(* PLC project Generated.project, CODESYS CODESYS V3.5 SP19 Patch 1 *)
(* stored: creationDateTime 2026-09-06T13:00:42.383652, modificationDateTime 2026-09-06T13:00:42.383652 *)

(* ======================================================================= 🧩 ST_Fault — Brique socle défaut (2 vues : live + latchée) ─────────────────────────────────────────────────────────────── 🎯 Rôle : porter l'état défaut d'un composant, applicable dans TOUS les cas (acquittable ou non), sans brique warning séparée. • Vue LIVE (Error / ErrorId) : suit la cause, retombe seule à 0. • Vue LATCHÉE (Latched / LatchedId): mémorisée au défaut, reste jusqu'au front Reset. Le choix acquittable / non-acquittable se fait PAR CAUSE (ST_FaultCause.Latching), jamais par bloc. 🔒 Sécurité : interlock TOUJOURS sur la cause brute (Error / ErrorId), jamais sur l'acquittement. Reset TOUJOURS effectif, jamais conditionné (std §9). 🧬 Composition : brique de base réutilisable — sortie de FB, struct métier, GVL. Texte IHM NON stocké ici : dérivé côté IHM depuis LatchedId / ErrorId. 📄 Doc : DOC/STDS/CODE_QUALITY_STANDARDS.md §2quinquies / §9 ======================================================================= *)
TYPE ST_Fault : STRUCT
  Error : BOOL;  (* <-- [DIAG] vue LIVE : au moins une cause présente maintenant *)
  ErrorId : WORD;  (* <-- [DIAG] bitfield des causes présentes maintenant (0 si aucune) *)
  Latched : BOOL;  (* <-- [DIAG] vue LATCHÉE : défaut non acquitté, reste jusqu'au front Reset *)
  LatchedId : WORD;  (* <-- [DIAG] ErrorId figé à l'apparition du défaut, effacé au Reset *)
END_STRUCT;
END_TYPE

(* ======================================================================= 🧩 ST_FaultCause — Cause élémentaire alimentant ST_Fault (socle FB_FaultCore) ─────────────────────────────────────────────────────────────── 🎯 Rôle : une cause exprimée EN CLAIR (BOOL + libellé), sans bitfield ni masque. Le FB métier remplit une liste (ARRAY[0..15] OF ST_FaultCause) ; le socle FB_FaultCore en déduit ST_Fault (vue live + vue latchée). 🔒 Sécurité : interlock TOUJOURS sur Active (cause brute), jamais sur le latch. Latching = TRUE → la cause ARME la vue latchée (défaut à acquitter). Latching = FALSE → la cause n'alimente que la vue live (retombe seule). Fail-safe : une cause laissée à Latching=FALSE reste visible en live — pour la rendre acquittable, il faut le déclarer explicitement. 📄 Doc : DOC/STDS/CODE_QUALITY_STANDARDS.md §2quinquies / §9 ======================================================================= *)
TYPE ST_FaultCause : STRUCT
  Active : BOOL;  (* 1 = cause présente maintenant (interlock sur cette valeur) *)
  Latching : BOOL;  (* 1 = cause à acquitter (arme Latched) ; 0 = live seulement *)
  Texte : STRING;  (* libellé prêt IHM (non stocké dans ST_Fault, dérivé côté IHM) *)
END_STRUCT;
END_TYPE

(* ======================================================================= 🔌 FB_Encoder_Abs — Acquisition codeur absolu (accès bus EtherCAT) ─────────────────────────────────────────────────────────────── 🎯 Rôle : Accès bus EtherCAT, extraction positions brutes et séquence de Preset SDO 🔒 Polarité : EncoderAvailable=TRUE si communication bus et esclave OK 🔌 Architecture : Module d'acquisition codeur absolu 📄 Doc métier : DOC/AF/AF_Partie-09_Fonction_Encoder_v2.4.md ======================================================================= === DECLARATION (à coller dans la partie déclaration du POU FB_Encoder_Abs) === *)
FUNCTION_BLOCK FB_Encoder_Abs
  VAR_INPUT
    Enable : BOOL;  (* === COMMANDES & AUTORISATIONS === --> [CMD] Autorisation generale FB (TRUE=Autorise) *)
    Reset : BOOL;  (* --> [CMD] Acquittement defaut (front montant) *)
    PresetRequest : BOOL;  (* --> [CMD] Demande de preset (front montant) *)
    RawPosIn : UDINT;  (* === BUS ETHERCAT & CAPTEUR HW === --> [HW] Position brute EtherCAT *)
    AlarmsIn : UINT;  (* --> [HW] Codes alarmes bruts EtherCAT *)
    WarningsIn : UINT;  (* --> [HW] Codes avertissements bruts EtherCAT *)
    SlaveOperational : BOOL;  (* --> [HW] Statut esclave EtherCAT operationnel *)
    PointsPerRev : UDINT := 8192;  (* === PARAMETRES & REGLAGES === --> [CFG] Resolution codeur (pts/tour) *)
    PresetValue : UDINT;  (* --> [CFG] Valeur cible de preset *)
    PresetTimeout : TIME := TIME#2s0ms;  (* --> [CFG] Temporisation max attente preset *)
    PresetTolerancePts : UDINT := 10;  (* --> [CFG] Tolerance relecture post-preset (pts) *)
  END_VAR
  VAR_OUTPUT
    Ready : BOOL;  (* === ETATS IEC & SYNOPTIQUE === <-- [STAT] FB pret a fonctionner *)
    Fault : ST_Fault;  (* 🧩 Statut transverse (forme cible ST_Fault) *)
    RawPos : UDINT;  (* === MESURES & DONNEES CODEUR === <-- [DIAG] Position brute gelee si non disponible *)
    EncoderAvailable : BOOL;  (* <-- [STAT] Codeur operationnel et disponible *)
    AngleRaw : UINT;  (* <-- [DIAG] Angle brut sur un tour (MOD PointsPerRev) *)
    TurnCount : UDINT;  (* <-- [DIAG] Nombre de tours bruts (RawPos / PointsPerRev) *)
    PresetTriggerCmd : WORD;  (* === COMMANDES & ECHANGE BUS ETHERCAT === <-- [ACT] Ordre declenchement preset vers PDO Rx *)
    CodeSeqTriggerCmd : WORD;  (* <-- [ACT] Ordre sequence code vers PDO Rx *)
    PresetValueOut : UDINT;  (* <-- [ACT] Valeur de preset transmise au PDO Rx *)
  END_VAR
  VAR
    ResetEdge : R_TRIG;  (* === DETECTEURS DE FRONT === . [LOC] Detecteur front montant Reset *)
    PresetReqEdge : R_TRIG;  (* . [LOC] Detecteur front montant PresetRequest *)
    PresetTimer : TON;  (* === TEMPORISATEURS INTERNES === . [LOC] Temporisateur timeout sequence preset *)
    PresetTimerVisual : TON;  (* . [LOC] Temporisateur maintien visuel impulsion (500ms) *)
    PresetSeqStep : INT;  (* === VARIABLES INTERNES DE CALCUL & ETAT === . [LOC] Etape sequence preset (0:IDLE, 1:PULSE/WAIT) *)
    RawDiff : DINT;  (* . [LOC] Ecart signe entre RawPos et PresetValueOut *)
    PresetCompleted : BOOL;  (* . [LOC] Fait de fin de maintien preset (un scan) *)
    PresetTimeoutError : BOOL;  (* . [LOC] Latch interne timeout séquence preset *)
    instFault : FB_FaultCore;  (* === SOCLE DEFAUT (FB_FaultCore) === * [INST] Socle défaut transverse *)
    instCauses : ARRAY[0..15] OF ST_FaultCause;  (* . [LOC] Table des causes nommées *)
  END_VAR

            

// === IMPLEMENTATION (à coller dans le corps ST du POU FB_Encoder_Abs) ===

{region "§1 Causes & Socle Défaut (évalué en continu)"}
// 🔑 1. RESET FRONT
ResetEdge(CLK := Reset);

// 🔍 2. DIAGNOSTIC BUS / ALARME (Cause 0 : live)
instCauses[0].Active   := (AlarmsIn <> 0) OR NOT SlaveOperational;
instCauses[0].Latching := FALSE;
instCauses[0].Texte    := 'Defaut communication EtherCAT codeur absolu';

// ⏱️ 3. TIMEOUT PRESET (Cause 1 : latched)
IF ResetEdge.Q AND (PresetSeqStep = 0) THEN
    PresetTimeoutError := FALSE;
END_IF;
instCauses[1].Active   := PresetTimeoutError;
instCauses[1].Latching := TRUE;
instCauses[1].Texte    := 'Timeout sequence preset SDO codeur';

// Appel du socle de défaut
instFault(Enable := Enable, Reset := Reset, Causes := instCauses);
Fault := instFault.Fault;

EncoderAvailable := NOT instCauses[0].Active;
{endregion}

{region "§2 Gate neutralisation"}
// 🛑 2. GATE
IF NOT Enable THEN
    EncoderAvailable := FALSE;
    Ready := FALSE;
    PresetTriggerCmd := 0; CodeSeqTriggerCmd := 0; PresetValueOut := 0;
    PresetSeqStep := 0;
    PresetCompleted := FALSE;
    PresetTimer(IN := FALSE, PT := PresetTimeout);
    PresetTimerVisual(IN := FALSE, PT := T#500MS);
    // RawPos, AngleRaw et TurnCount sont volontairement gelés hors Enable
    // (AF09 F09.01 / AC5) : aucune lecture bus ni remise a zero dans ce gate.
    RETURN;
END_IF;

Ready := Enable AND NOT Fault.Latched;
{endregion}

{region "§3 Lecture position"}
// 📥 3. LECTURE POSITION — GELER SUR DOUTE (Partie10 §6)
// Si EncoderAvailable=FALSE : RawPos/AngleRaw/TurnCount conservent leur dernière valeur (pas de RETURN
// global ici pour ne pas geler aussi la séquence preset/l'état — seule la lecture est gelée).
IF EncoderAvailable THEN
    RawPos := RawPosIn;   // Sens de comptage géré côté codeur (CoE 6000h bit0, startup parameter CODESYS) — voir Partie10 §3bis. Plus de calcul ici.
    AngleRaw := UDINT_TO_UINT(RawPos MOD PointsPerRev);
    TurnCount := RawPos / PointsPerRev;
END_IF;
{endregion}

{region "§4 Séquence preset"}
// 🔧 4. SÉQUENCE PRESET (écriture bus)
// PresetTriggerCmd := 2 déclenche le référencement à PresetValue (valeur de commande, pas un
// masque de bits). CodeSeqTriggerCmd : rôle non identifié — laissé à 0, PAS piloté tant que sa
// fonction n'est pas confirmée. Ne jamais lui donner une valeur arbitraire.
PresetReqEdge(CLK := PresetRequest);
PresetCompleted := FALSE;
CodeSeqTriggerCmd := 0;                 // non piloté — rôle inconnu, voir note ci-dessus
CASE PresetSeqStep OF
    0: // IDLE
        PresetTriggerCmd := 0;
        IF PresetReqEdge.Q AND EncoderAvailable THEN
            PresetValueOut := PresetValue;
            PresetSeqStep := 1;
            PresetTimer(IN := TRUE, PT := PresetTimeout);
        END_IF;
    1: // Déclenchement preset (laissé actif pendant 0.5s pour confort visuel en simulation/bus)
        PresetTriggerCmd := 2;   // Référence le codeur à PresetValueOut
        RawDiff := UDINT_TO_DINT(RawPos) - UDINT_TO_DINT(PresetValueOut);
        IF ABS(RawDiff) <= UDINT_TO_DINT(PresetTolerancePts) THEN
            PresetTimer(IN := FALSE, PT := PresetTimeout);
            PresetTimerVisual(IN := TRUE, PT := T#500MS);
            IF PresetTimerVisual.Q THEN
                PresetTriggerCmd := 0;
                PresetCompleted := TRUE;
                PresetSeqStep := 0;
                PresetTimerVisual(IN := FALSE, PT := T#500MS);
            END_IF;
        ELSIF PresetTimer.Q THEN
            PresetTriggerCmd := 0;
            PresetTimeoutError := TRUE;
            PresetSeqStep := 0;
            PresetTimer(IN := FALSE, PT := PresetTimeout);
            PresetTimerVisual(IN := FALSE, PT := T#500MS);
        END_IF;
END_CASE;
{endregion}

          
END_FUNCTION_BLOCK

(* ======================================================================= 🧩 FB_FaultCore — Socle de remplissage de ST_Fault (vue live + vue latchée) ─────────────────────────────────────────────────────────────── 🎯 Rôle : à partir d'une LISTE de causes en clair (ARRAY[0..15] OF ST_FaultCause), produire la brique ST_Fault : • Error / ErrorId : vue LIVE, suit les causes Active, retombe seule. • Latched / LatchedId: vue LATCHÉE, chaque bit figé à l'apparition d'une cause `Active AND Latching`, conservé jusqu'au front Reset. 🔒 Sécurité : - interlock TOUJOURS sur `Causes[i].Active` (cause brute), jamais sur le latch. - Reset TOUJOURS effectif, jamais conditionné (std §9) — agit même Enable=FALSE. - Latching=FALSE → cause visible en LIVE seulement (fail-safe : reste visible). - un défaut laté non acquitté reste publié même FB désactivé (pas d'effacement silencieux sur bascule Enable OFF→ON sans Reset). - une cause à acquitter réapparue re-arme son bit (ré-alarme). 🧬 Un seul socle, réutilisé par tout FB `standard` qui expose un ST_Fault. Pas de State, pas de Warning, pas de texte — hors périmètre de ce socle. 📄 Doc : DOC/STDS/CODE_QUALITY_STANDARDS.md §2quinquies / §9 ======================================================================= *)
FUNCTION_BLOCK FB_FaultCore
  VAR_INPUT
    Enable : BOOL;  (* --> [CMD] Autorisation générale du FB porteur *)
    Reset : BOOL;  (* --> [CMD] Front d'acquittement (jamais conditionné, §9) *)
    Causes : ARRAY[0..15] OF ST_FaultCause;  (* --> [CMD] Liste des causes en clair (Active / Latching / Texte) *)
  END_VAR
  VAR_OUTPUT
    Ready : BOOL;  (* <-- [STAT] FB porteur autorisé (= Enable) *)
    Fault : ST_Fault;  (* <-- [DIAG] Brique défaut (mappée 1:1 sur la sortie du FB porteur) *)
  END_VAR
  VAR
    ResetEdge : R_TRIG;  (* . [LOC] Front montant Reset *)
    Latch : ARRAY[0..15] OF BOOL;  (* . [LOC] Bit laté par cause, jusqu'au Reset *)
    i : INT;  (* . [LOC] Index de parcours de la liste *)
  END_VAR

            

{region "§1 Reset (front, toujours effectif)"}
// Front Reset : efface tous les latches. Jamais conditionné, agit même Enable=FALSE (§9).
Ready := Enable;
ResetEdge(CLK := Reset);
IF ResetEdge.Q THEN
    FOR i := 0 TO 15 DO Latch[i] := FALSE; END_FOR;
END_IF;
{endregion}

{region "§2 Vue LIVE — Error / ErrorId"}
// Bitfield des causes présentes MAINTENANT. Retombe seule à 0 quand les causes disparaissent.
// Non évaluée si Enable=FALSE (pas de lecture de cause hors autorisation).
Fault.ErrorId := 0;
IF Enable THEN
    FOR i := 0 TO 15 DO
        IF Causes[i].Active THEN
            Fault.ErrorId := Fault.ErrorId OR SHL(WORD#1, INT_TO_DWORD(i));
        END_IF;
    END_FOR;
END_IF;
Fault.Error := (Fault.ErrorId <> 0);
{endregion}

{region "§3 Armement des latches (causes à acquitter)"}
// Une cause Active ET Latching arme son bit ; le bit reste jusqu'au front Reset (§1),
// même si la cause disparaît. Réapparition => ré-armement (ré-alarme).
IF Enable THEN
    FOR i := 0 TO 15 DO
        IF Causes[i].Active AND Causes[i].Latching THEN
            Latch[i] := TRUE;
        END_IF;
    END_FOR;
END_IF;
{endregion}

{region "§4 Vue LATCHÉE — Latched / LatchedId"}
// Toujours publiée, y compris Enable=FALSE : un défaut non acquitté reste visible.
Fault.LatchedId := 0;
FOR i := 0 TO 15 DO
    IF Latch[i] THEN
        Fault.LatchedId := Fault.LatchedId OR SHL(WORD#1, INT_TO_DWORD(i));
    END_IF;
END_FOR;
Fault.Latched := (Fault.LatchedId <> 0);
{endregion}

          
END_FUNCTION_BLOCK
